	                #sFB_PECUpdate_380(iUDT_PECUpdateConfiguration := #iUDT_Configuration."380".PEC_Eos,
	                                   iUDT_ConveyorCommonConfiguration := #iUDT_Configuration."380".Conveyor.Common,
	                                   ix_PEC := #iUDT_MotorInput380.AllSensorPortInputs.LeftSensor,
	                                   ix_TeachingMode := FALSE,
	                                   qUDT_Status => #iqUDT_WorkstationStatus."380".PEC_Eos,
	                                   qi_GINwrite => #ti_dummy,
	                                   qx_PECFiltered => #tx_dummy,
	                                   iqa_TrackingData := #sa_TrackingArray_380,
	                                   iqUDT_ConveyorInterface := #sUDT_Interface_380,
	                                   iqUDT_UnknownGINRange := #iqUDT_UnknownGINRange,
	                                   iqUDT_FifoHeader := "DB_FIFOLostGIN".Header,
	                                   iqa_FifoData := "DB_FIFOLostGIN".Data,
	                                   iqUDT_Statistics := #iqUDT_WorkstationStatistics."380".PEC_Eos);

	            END_REGION

	            REGION Conveyor

	                #sUDT_Handshake_380.RTR := #iqUDT_WorkstationStatus."380".PEC_Eos.PEC;

	                #sFB_Conveyor_380(iUDT_ConveyorConfiguration := #iUDT_Configuration."380".Conveyor,
	                                  idi_PECEoSDistance := #iUDT_Configuration."380".PEC_Eos.Distance,
	                                  idi_PECBoSDistance := 0,
	                                  ii_ExternalSpeed := 0,
	                                  ix_SafetyOk := #ix_SafetyOk,
	                                  ix_24vOk := #ix_24vOk,
	                                  ix_400vOk := #ix_400vOk,
	                                  ix_HardwareOk := #ix_HardwareOk,
	                                  ix_ReverseDirection := #sx_DirectionChange380,
	                                  ix_PECEoS := #iqUDT_WorkstationStatus."380".PEC_Eos.PEC,
	                                  ix_PECBoS := TRUE,
	                                  ix_ExternalRequestHold := false,
	                                  qUDT_HMIStatus => #iqUDT_WorkstationStatus."380".Conveyor,
	                                  qUDT_Status => #iqUDT_WorkstationCommonStatus."380",
	                                  iqUDT_EquipmentControl := #iqUDT_EquipmentControl,
	                                  iqUDT_ConveyorCommand := #iqUDT_WorkstationCommands."380".Conveyor,
	                                  iqUDT_ConveyorInterface := #sUDT_Interface_380,
	                                  iqUDT_HandShakeUp := #sUDT_Handshake_360,
	                                  iqUDT_HandShake := #sUDT_Handshake_380,
	                                  iqUDT_Statistics := #iqUDT_WorkstationStatistics."380".Conveyor);
	            END_REGION

	            REGION MCO
	                #sFB_MCOConveyLinxAixController_380(iUDT_AixConfig := #iUDT_Configuration."380".MCO_M01,
	                                                    iv_AixInputsModule := #iUDT_MotorInput380,
	                                                    ix_24vOk := #ix_24vOk,
	                                                    ix_SimulationModeActive := "DB_Memory".Simulation,
	                                                    ii_MotorPositionId := 1,
	                                                    qUDT_HMIStatus => #iqUDT_WorkstationStatus."380".MCO_M01,
	                                                    iqv_AixOutputsModule := #qUDT_MotorOutput380,
	                                                    iqUDT_ConveyorInterface := #sUDT_Interface_380,
	                                                    iqUDT_MCOStatistics := #iqUDT_WorkstationStatistics."380".MCO_M01);
	            END_REGION


	        END_REGION

	        REGION 390

	            REGION Displacement

	                #sFB_Displacement390(#sUDT_Interface_390);

	            END_REGION

	            REGION Tracking

	                #sFB_Tracking_390(iUDT_ConveyorCommonConfiguration := #iUDT_Configuration."390".Conveyor.Common,
	                                  iqa_TrackingData := #sa_TrackingArray_390,
	                                  iqUDT_ConveyorInterface := #sUDT_Interface_390,
	                                  iqUDT_HandshakeUp := #sUDT_Handshake_370,
	                                  iqUDT_Handshake := #sUDT_Handshake_390);
	            END_REGION

	            REGION EOS

	                #sFB_PECUpdate_390(iUDT_PECUpdateConfiguration := #iUDT_Configuration."390".PEC_Eos,
	                                   iUDT_ConveyorCommonConfiguration := #iUDT_Configuration."390".Conveyor.Common,
	                                   ix_PEC := #iUDT_MotorInput390.AllSensorPortInputs.LeftSensor,
	                                   ix_TeachingMode := FALSE,
	                                   qUDT_Status => #iqUDT_WorkstationStatus."390".PEC_Eos,
	                                   qi_GINwrite => #ti_dummy,
	                                   qx_PECFiltered => #tx_dummy,
	                                   iqa_TrackingData := #sa_TrackingArray_390,
	                                   iqUDT_ConveyorInterface := #sUDT_Interface_390,
	                                   iqUDT_UnknownGINRange := #iqUDT_UnknownGINRange,
	                                   iqUDT_FifoHeader := "DB_FIFOLostGIN".Header,
	                                   iqa_FifoData := "DB_FIFOLostGIN".Data,
	                                   iqUDT_Statistics := #iqUDT_WorkstationStatistics."390".PEC_Eos);

	            END_REGION

	            REGION Conveyor

	                #sUDT_Handshake_390.RTR := #iqUDT_WorkstationStatus."390".PEC_Eos.PEC;


	                #sFB_Conveyor_390(iUDT_ConveyorConfiguration := #iUDT_Configuration."390".Conveyor,
	                                  idi_PECEoSDistance := #iUDT_Configuration."390".PEC_Eos.Distance,
	                                  idi_PECBoSDistance := 0,
	                                  ii_ExternalSpeed := 0,
	                                  ix_SafetyOk := #ix_SafetyOk,
	                                  ix_24vOk := #ix_24vOk,
	                                  ix_400vOk := #ix_400vOk,
	                                  ix_HardwareOk := #ix_HardwareOk,
	                                  ix_ReverseDirection := #sx_DirectionChange390,
	                                  ix_PECEoS := #iqUDT_WorkstationStatus."390".PEC_Eos.PEC,
	                                  ix_PECBoS := TRUE,
	                                  ix_ExternalRequestHold := FALSE,
	                                  qUDT_HMIStatus => #iqUDT_WorkstationStatus."390".Conveyor,
	                                  qUDT_Status => #iqUDT_WorkstationCommonStatus."390",
	                                  iqUDT_EquipmentControl := #iqUDT_EquipmentControl,
	                                  iqUDT_ConveyorCommand := #iqUDT_WorkstationCommands."390".Conveyor,
	                                  iqUDT_ConveyorInterface := #sUDT_Interface_390,
	                                  iqUDT_HandShakeUp := #sUDT_Handshake_370,
	                                  iqUDT_HandShake := #sUDT_Handshake_390,
	                                  iqUDT_Statistics := #iqUDT_WorkstationStatistics."390".Conveyor);
	            END_REGION

	            REGION MCO
	                #sFB_MCOConveyLinxAixController_390(iUDT_AixConfig := #iUDT_Configuration."390".MCO_M01,
	                                                    iv_AixInputsModule := #iUDT_MotorInput390,
	                                                    ix_24vOk := #ix_24vOk,
	                                                    ix_SimulationModeActive := "DB_Memory".Simulation,
	                                                    ii_MotorPositionId := 1,
	                                                    qUDT_HMIStatus => #iqUDT_WorkstationStatus."390".MCO_M01,
	                                                    iqv_AixOutputsModule := #qUDT_MotorOutput390,
	                                                    iqUDT_ConveyorInterface := #sUDT_Interface_390,
	                                                    iqUDT_MCOStatistics := #iqUDT_WorkstationStatistics."390".MCO_M01);
	            END_REGION


	        END_REGION
	        REGION 230

	            REGION Displacement

	                #sFB_Displacement230(#sUDT_Interface_230);

	            END_REGION

	            REGION Tracking

	                #sFB_Tracking_230(iUDT_ConveyorCommonConfiguration := #iUDT_Configuration."230".Conveyor.Common,
	                                  iqa_TrackingData := #sa_TrackingArray_230,
	                                  iqUDT_ConveyorInterface := #sUDT_Interface_230,
	                                  iqUDT_HandshakeUp := #sUDT_Handshake_230,
	                                  iqUDT_Handshake := #sUDT_Handshake_230);
	            END_REGION

	            REGION EOS

	                #sFB_PECUpdate_230(iUDT_PECUpdateConfiguration := #iUDT_Configuration."230".PEC_Eos,
	                                   iUDT_ConveyorCommonConfiguration := #iUDT_Configuration."230".Conveyor.Common,
	                                   ix_PEC := #iUDT_MotorInput230.AllSensorPortInputs.LeftSensor,
	                                   ix_TeachingMode := FALSE,
	                                   qUDT_Status => #iqUDT_WorkstationStatus."230".PEC_Eos,
	                                   qi_GINwrite => #ti_dummy,
	                                   qx_PECFiltered => #tx_dummy,
	                                   iqa_TrackingData := #sa_TrackingArray_230,
	                                   iqUDT_ConveyorInterface := #sUDT_Interface_230,
	                                   iqUDT_UnknownGINRange := #iqUDT_UnknownGINRange,
	                                   iqUDT_FifoHeader := "DB_FIFOLostGIN".Header,
	                                   iqa_FifoData := "DB_FIFOLostGIN".Data,
	                                   iqUDT_Statistics := #iqUDT_WorkstationStatistics."230".PEC_Eos);

	            END_REGION

	            REGION Conveyor
	                #sUDT_Handshake_230.RTR := #sUDT_Handshake_230.RTR OR #iqUDT_WorkstationStatus."230".PEC_Eos.PEC;

	                #sFB_Conveyor_230(iUDT_ConveyorConfiguration := #iUDT_Configuration."230".Conveyor,
	                                  idi_PECEoSDistance := #iUDT_Configuration."230".PEC_Eos.Distance,
	                                  idi_PECBoSDistance := 0,
	                                  ii_ExternalSpeed := 0,
	                                  ix_SafetyOk := #ix_SafetyOk,
	                                  ix_24vOk := #ix_24vOk,
	                                  ix_400vOk := #ix_400vOk,
	                                  ix_HardwareOk := #ix_HardwareOk,
	                                  ix_PECEoS := #iqUDT_WorkstationStatus."230".PEC_Eos.PEC,
	                                  ix_PECBoS := TRUE,
	                                  ix_ExternalRequestHold := #sx_Hold230,
	                                  qUDT_HMIStatus => #iqUDT_WorkstationStatus."230".Conveyor,
	                                  qUDT_Status => #iqUDT_WorkstationCommonStatus."230",
	                                  iqUDT_EquipmentControl := #iqUDT_EquipmentControl,
	                                  iqUDT_ConveyorCommand := #iqUDT_WorkstationCommands."230".Conveyor,
	                                  iqUDT_ConveyorInterface := #sUDT_Interface_230,
	                                  iqUDT_HandShakeUp := #sUDT_Handshake_230,
	                                  iqUDT_HandShake := #sUDT_Handshake_230,
	                                  iqUDT_Statistics := #iqUDT_WorkstationStatistics."230".Conveyor);
	            END_REGION

	            REGION MCO
	                #sFB_MCOConveyLinxAixController_230(iUDT_AixConfig := #iUDT_Configuration."230".MCO_M01,
	                                                    iv_AixInputsModule := #iUDT_MotorInput230,
	                                                    ix_24vOk := #ix_24vOk,
	                                                    ix_SimulationModeActive := "DB_Memory".Simulation,
	                                                    ii_MotorPositionId := 1,
	                                                    qUDT_HMIStatus => #iqUDT_WorkstationStatus."230".MCO_M01,
	                                                    iqv_AixOutputsModule := #qUDT_MotorOutput230,
	                                                    iqUDT_ConveyorInterface := #sUDT_Interface_230,
	                                                    iqUDT_MCOStatistics := #iqUDT_WorkstationStatistics."230".MCO_M01);
	            END_REGION

	        END_REGION

	        REGION 240

	            REGION Displacement

	                #sFB_Displacement240(#sUDT_Interface_240);

	            END_REGION

	            REGION MCO
	                #sFB_MCOConveyLinxAixController_240(iUDT_AixConfig := #iUDT_Configuration."240".MCO_M01,
	                                                    iv_AixInputsModule := #iUDT_MotorInput240,
	                                                    ii_PositionSetpoint := #iqUDT_RATPositioning240.Lower.EndPosition,
	                                                    ix_24vOk := #ix_24vOk,
	                                                    ix_SimulationModeActive := "DB_Memory".Simulation,
	                                                    ii_MotorPositionId := 1,
	                                                    ix_StartPositioning := #iqUDT_RATPositioning240.Lower.Start,
	                                                    ix_ResetPosition := #iqUDT_RATPositioning240.Lower.ResetPosition,
	                                                    qUDT_HMIStatus => #iqUDT_WorkstationStatus."240".MCO_M01,
	                                                    qx_Positioned => #iqUDT_RATPositioning240.Lower.Done,
	                                                    iqv_AixOutputsModule := #qUDT_MotorOutput240,
	                                                    iqUDT_ConveyorInterface := #sUDT_Interface_240,
	                                                    iqUDT_MCOStatistics := #iqUDT_WorkstationStatistics."240".MCO_M01);
	            END_REGION


	        END_REGION

	        REGION 241

	            REGION Displacement

	                #sFB_Displacement241(#sUDT_Interface_241);

	            END_REGION

	            REGION RAT

	                #sFB_RightAngledTransfer_241(iUDT_Configuration := #iUDT_Configuration."241".RightAngledTransfer,
	                                             iUDT_LowerConveyorConfiguration := #iUDT_Configuration."240".Conveyor,
	                                             iUDT_UpperConveyorConfiguration := #iUDT_Configuration."241".Conveyor,
	                                             iUDT_PECConfiguration := #iUDT_Configuration."240".PEC_Eos,
	                                             ii_DestinationA := #si_240DestinationA,
	                                             ii_DestinationB := #si_240DestinationB,
	                                             ii_DestinationC := #si_240DestinationC,
	                                             ii_DestinationD := #si_240DestinationD,
	                                             ix_HardwareOk := #ix_HardwareOk,
	                                             ix_400vOk := #ix_400vOk,
	                                             ix_24vOk := #ix_24vOk,
	                                             ix_SafetyOk := #ix_SafetyOk,
	                                             ix_AirPressureOk := #ix_AirPressureOk,
	                                             ix_SectionIsDown := #ix_SectionIsDown241,
	                                             ix_SectionIsUp := #ix_SectionIsUp241,
	                                             ix_ConveyorAAuto := #iqUDT_WorkstationCommonStatus."230".AutoON,
	                                             ix_ConveyorBAuto := #iqUDT_WorkstationCommonStatus."250".AutoON,
	                                             ix_ConveyorCAuto := FALSE,
	                                             ix_ConveyorDAuto := #iqUDT_WorkstationCommonStatus."370".AutoON,
	                                             ix_PEC := #iUDT_MotorInput240.AllSensorPortInputs.LeftSensor,
	                                             ix_ExternalReceiveRequestA := NOT #iqUDT_WorkstationStatus."230".PEC_Eos.PEC AND NOT #sx_TransferOut380 AND NOT #sx_TransferOut390,
	                                             ix_ExternalReceiveRequestB := false,
	                                             ix_ExternalReceiveRequestC := false,
	                                             ix_ExternalReceiveRequestD := #sFB_RightAngledTransfer_371.qx_ExternalSendRequestD,//NOT #iUDT_MotorInput370.AllSensorPortInputs.LeftSensor AND (#sx_TransferOut380 OR #sx_TransferOut390 OR #iqx_ClearRightStation),,
	                                             ix_PECInfeedA := #iqUDT_WorkstationStatus."230".PEC_Eos.PEC,
	                                             ix_PECInfeedD := #iqUDT_WorkstationStatus."370".PEC_Eos.PEC,
	                                             qUDT_HMIRATStatus => #iqUDT_WorkstationStatus."241".RightAngledTransfer,
	                                             qUDT_HMIConveyorStatus => #iqUDT_WorkstationStatus."240".Conveyor,
	                                             qUDT_HMIPECStatus => #iqUDT_WorkstationStatus."240".PEC_Eos,
	                                             qUDT_RATStatus => #iqUDT_WorkstationCommonStatus."241",
	                                             qUDT_ConveyorStatus => #iqUDT_WorkstationCommonStatus."240",
	                                             qx_PopupControl => #qx_PopupControl241,
	                                             iqUDT_EquipmentControl := #iqUDT_EquipmentControl,
	                                             iqUDT_RATCommand := #iqUDT_WorkstationCommands."241".RightAngledTransfer,
	                                             iqUDT_ConveyorCommand := #iqUDT_WorkstationCommands."240".Conveyor,
	                                             iqUDT_RATStatistics := #iqUDT_WorkstationStatistics."241".RightAngledTransfer,
	                                             iqUDT_ConveyorStatistics := #iqUDT_WorkstationStatistics."240".Conveyor,
	                                             iqUDT_PECStatistics := #iqUDT_WorkstationStatistics."240".PEC_Eos,
	                                             iqUDT_HandShakeConveyorA := #sUDT_Handshake_230,
	                                             iqUDT_HandShakeConveyorB := #sUDT_Handshake_240,
	                                             iqUDT_HandShakeConveyorC := #sUDT_Handshake_241,
	                                             iqUDT_HandShakeConveyorD := #sUDT_Handshake_371,
	                                             iqUDT_LowerConveyorInterface := #sUDT_Interface_240,
	                                             iqUDT_UpperConveyorInterface := #sUDT_Interface_241,
	                                             iqUDT_RATPositioning := #iqUDT_RATPositioning240,
	                                             iqUDT_BladeStopEoSInterface := #tUDT_DummyBladeStop,
	                                             iqUDT_BladeStopBoSInterface := #tUDT_DummyBladeStop);

	            END_REGION

	            REGION MCO
	                #sFB_MCOConveyLinxAixController_241(iUDT_AixConfig := #iUDT_Configuration."241".MCO_M01,
	                                                    iv_AixInputsModule := #iUDT_MotorInput240,
	                                                    ii_PositionSetpoint := #iqUDT_RATPositioning240.Upper.EndPosition,
	                                                    ix_24vOk := #ix_24vOk,
	                                                    ix_SimulationModeActive := "DB_Memory".Simulation,
	                                                    ii_MotorPositionId := 2,
	                                                    ix_StartPositioning := #iqUDT_RATPositioning240.Upper.Start,
	                                                    ix_ResetPosition := #iqUDT_RATPositioning240.Upper.ResetPosition,
	                                                    qUDT_HMIStatus => #iqUDT_WorkstationStatus."241".MCO_M01,
	                                                    qx_Positioned => #iqUDT_RATPositioning240.Upper.Done,
	                                                    iqv_AixOutputsModule := #qUDT_MotorOutput240,
	                                                    iqUDT_ConveyorInterface := #sUDT_Interface_241,
	                                                    iqUDT_MCOStatistics := #iqUDT_WorkstationStatistics."241".MCO_M01);
	            END_REGION
	        END_REGION

	        REGION 250

	            REGION Displacement

	                #sFB_Displacement250(#sUDT_Interface_250);

	            END_REGION

	            REGION EOS

	                #sFB_PECUpdate_250(iUDT_PECUpdateConfiguration := #iUDT_Configuration."250".PEC_EoS,
	                                   iUDT_ConveyorCommonConfiguration := #iUDT_Configuration."250".Conveyor.Common,
	                                   ix_PEC := #iUDT_MotorInput250.AllSensorPortInputs.LeftSensor,
	                                   ix_TeachingMode := FALSE,
	                                   qUDT_Status => #iqUDT_WorkstationStatus."250".PEC_EoS,
	                                   qi_GINwrite => #ti_dummy,
	                                   qx_PECFiltered => #tx_dummy,
	                                   iqa_TrackingData := #sa_TrackingArray_250,
	                                   iqUDT_ConveyorInterface := #sUDT_Interface_250,
	                                   iqUDT_UnknownGINRange := #iqUDT_UnknownGINRange,
	                                   iqUDT_FifoHeader := "DB_FIFOLostGIN".Header,
	                                   iqa_FifoData := "DB_FIFOLostGIN".Data,
	                                   iqUDT_Statistics := #iqUDT_WorkstationStatistics."250".PEC_EoS);

	            END_REGION

	            REGION Conveyor

	                #sUDT_Handshake_250.RTR := #sUDT_Handshake_250.RTR OR #iqUDT_WorkstationStatus."250".PEC_EoS.PEC;

	                #sFB_Conveyor_250(iUDT_ConveyorConfiguration := #iUDT_Configuration."250".Conveyor,
	                                  idi_PECEoSDistance := #iUDT_Configuration."250".PEC_EoS.Distance,
	                                  idi_PECBoSDistance := 0,
	                                  ii_ExternalSpeed := 0,
	                                  ix_SafetyOk := #ix_SafetyOk,
	                                  ix_24vOk := #ix_24vOk,
	                                  ix_400vOk := #ix_400vOk,
	                                  ix_HardwareOk := #ix_HardwareOk,
	                                  ix_PECEoS := #iqUDT_WorkstationStatus."250".PEC_EoS.PEC,
	                                  ix_PECBoS := TRUE,
	                                  ix_ExternalRequestHold := false,
	                                  qUDT_HMIStatus => #iqUDT_WorkstationStatus."250".Conveyor,
	                                  qUDT_Status => #iqUDT_WorkstationCommonStatus."250",
	                                  iqUDT_EquipmentControl := #iqUDT_EquipmentControl,
	                                  iqUDT_ConveyorCommand := #iqUDT_WorkstationCommands."250".Conveyor,
	                                  iqUDT_ConveyorInterface := #sUDT_Interface_250,
	                                  iqUDT_HandShakeUp := #sUDT_Handshake_240,
	                                  iqUDT_HandShake := #sUDT_Handshake_250,
	                                  iqUDT_Statistics := #iqUDT_WorkstationStatistics."250".Conveyor);
	            END_REGION

	            REGION MCO
	                #sFB_MCOConveyLinxAixController_250(iUDT_AixConfig := #iUDT_Configuration."250".MCO_M01,
	                                                    iv_AixInputsModule := #iUDT_MotorInput250,
	                                                    ix_24vOk := #ix_24vOk,
	                                                    ix_SimulationModeActive := "DB_Memory".Simulation,
	                                                    ii_MotorPositionId := 1,
	                                                    qUDT_HMIStatus => #iqUDT_WorkstationStatus."250".MCO_M01,
	                                                    iqv_AixOutputsModule := #qUDT_MotorOutput250,
	                                                    iqUDT_ConveyorInterface := #sUDT_Interface_250,
	                                                    iqUDT_MCOStatistics := #iqUDT_WorkstationStatistics."250".MCO_M01);
	            END_REGION


	        END_REGION

	        REGION 260


	            REGION Displacement

	                #sFB_Displacement260(#sUDT_Interface_260);

	            END_REGION

	            REGION Conveyor
	                #sFB_Conveyor_260(iUDT_ConveyorConfiguration := #iUDT_Configuration."260".Conveyor,
	                                  idi_PECEoSDistance := 0,
	                                  idi_PECBoSDistance := 0,
	                                  ii_ExternalSpeed := 0,
	                                  ix_SafetyOk := #ix_SafetyOk,
	                                  ix_24vOk := #ix_24vOk,
	                                  ix_400vOk := #ix_400vOk,
	                                  ix_HardwareOk := #ix_HardwareOk,
	                                  ix_PECEoS := TRUE,
	                                  ix_PECBoS := TRUE,
	                                  ix_ExternalRequestHold := false,
	                                  qUDT_HMIStatus => #iqUDT_WorkstationStatus."260".Conveyor,
	                                  qUDT_Status => #iqUDT_WorkstationCommonStatus."260",
	                                  iqUDT_EquipmentControl := #iqUDT_EquipmentControl,
	                                  iqUDT_ConveyorCommand := #iqUDT_WorkstationCommands."260".Conveyor,
	                                  iqUDT_ConveyorInterface := #sUDT_Interface_260,
	                                  iqUDT_HandShakeUp := #sUDT_Handshake_250,
	                                  iqUDT_HandShake := #sUDT_Handshake_260,
	                                  iqUDT_Statistics := #iqUDT_WorkstationStatistics."260".Conveyor);
	            END_REGION

	            REGION VFD

	                #sFB_VfdNORDPPO4_260(iUDT_VFDConfig := #iUDT_Configuration."260".VFD,
	                                     iUDT_VFDInputs := #iUDT_MotorInput260,
	                                     iUDT_MotorData := #iUDT_MotorData260,
	                                     ix_24vOk := #ix_24vOk,
	                                     ix_400vOk := #ix_400vOk,
	                                     ix_QuickStopDisable := TRUE,
	                                     ix_SimulationModeActive := "DB_Memory".Simulation,
	                                     qUDT_HMIStatus => #iqUDT_WorkstationStatus."260".VFD,
	                                     qUDT_VFDOutputs => #qUDT_MotorOutput260,
	                                     iqUDT_ConveyorInterface := #sUDT_Interface_260,
	                                     iqUDT_VFDStatistics := #iqUDT_WorkstationStatistics."260".VFD,
	                                     iqx_StartCommissioning := #iqx_StartComissioning260);

	            END_REGION


	        END_REGION

	        REGION 270

	            REGION Displacement

	                #sFB_Displacement270(#sUDT_Interface_270);

	            END_REGION

	            REGION EoS

	                #sFB_PEC_270(ix_PEC := #iUDT_MotorInput270.AllSensorPortInputs.LeftSensor,
	                             iUDT_PECConfiguration := #iUDT_Configuration."270".PEC_EoS,
	                             qUDT_HMIStatus => #iqUDT_WorkstationStatus."270".PEC_EoS,
	                             iqUDT_ConveyorInterface := #sUDT_Interface_270,
	                             iqUDT_PECStatistics := #iqUDT_WorkstationStatistics."270".PEC_EoS);

	            END_REGION

	            REGION Conveyor
	                #sFB_Conveyor_270(iUDT_ConveyorConfiguration := #iUDT_Configuration."270".Conveyor,
	                                  idi_PECEoSDistance := #iUDT_Configuration."270".PEC_EoS.Distance,
	                                  idi_PECBoSDistance := 0,
	                                  ii_ExternalSpeed := 0,
	                                  ix_SafetyOk := #ix_SafetyOk,
	                                  ix_24vOk := #ix_24vOk,
	                                  ix_400vOk := #ix_400vOk,
	                                  ix_HardwareOk := #ix_HardwareOk,
	                                  ix_PECEoS := #iqUDT_WorkstationStatus."270".PEC_EoS.PEC,
	                                  ix_PECBoS := TRUE,
	                                  ix_ExternalRequestHold := false,
	                                  qUDT_HMIStatus => #iqUDT_WorkstationStatus."270".Conveyor,
	                                  qUDT_Status => #iqUDT_WorkstationCommonStatus."270",
	                                  iqUDT_EquipmentControl := #iqUDT_EquipmentControl,
	                                  iqUDT_ConveyorCommand := #iqUDT_WorkstationCommands."270".Conveyor,
	                                  iqUDT_ConveyorInterface := #sUDT_Interface_270,
	                                  iqUDT_HandShakeUp := #sUDT_Handshake_260,
	                                  iqUDT_HandShake := #sUDT_Handshake_270,
	                                  iqUDT_Statistics := #iqUDT_WorkstationStatistics."270".Conveyor);
	            END_REGION

	            REGION MCO
	                #sFB_MCOConveyLinxAixController_270(iUDT_AixConfig := #iUDT_Configuration."270".MCO_M01,
	                                                    iv_AixInputsModule := #iUDT_MotorInput270,
	                                                    ix_24vOk := #ix_24vOk,
	                                                    ix_SimulationModeActive := "DB_Memory".Simulation,
	                                                    ii_MotorPositionId := 1,
	                                                    qUDT_HMIStatus => #iqUDT_WorkstationStatus."270".MCO_M01,
	                                                    iqv_AixOutputsModule := #qUDT_MotorOutput270,
	                                                    iqUDT_ConveyorInterface := #sUDT_Interface_270,
	                                                    iqUDT_MCOStatistics := #iqUDT_WorkstationStatistics."270".MCO_M01);
	            END_REGION
	        END_REGION

	        REGION 280

	            REGION Displacement

	                #sFB_Displacement280(#sUDT_Interface_280);

	            END_REGION

	            REGION EoS

	                #sFB_PEC_280(ix_PEC := #iUDT_MotorInput270.AllSensorPortInputs.RightSensor,
	                             iUDT_PECConfiguration := #iUDT_Configuration."280".PEC_EoS,
	                             qUDT_HMIStatus => #iqUDT_WorkstationStatus."280".PEC_EoS,
	                             iqUDT_ConveyorInterface := #sUDT_Interface_280,
	                             iqUDT_PECStatistics := #iqUDT_WorkstationStatistics."280".PEC_EoS);

	            END_REGION

	            REGION Conveyor
	                #iqUDT_HandshakeDownstream280.RTR := #iqUDT_HandshakeDownstream280.RTR OR #iqUDT_WorkstationStatus."280".PEC_EoS.PEC;
	                #sFB_Conveyor_280(iUDT_ConveyorConfiguration := #iUDT_Configuration."280".Conveyor,
	                                  idi_PECEoSDistance := #iUDT_Configuration."280".PEC_EoS.Distance,
	                                  idi_PECBoSDistance := 0,
	                                  ii_ExternalSpeed := 0,
	                                  ix_SafetyOk := #ix_SafetyOk,
	                                  ix_24vOk := #ix_24vOk,
	                                  ix_400vOk := #ix_400vOk,
	                                  ix_HardwareOk := #ix_HardwareOk,
	                                  ix_PECEoS := #iqUDT_WorkstationStatus."280".PEC_EoS.PEC,
	                                  ix_PECBoS := TRUE,
	                                  ix_ExternalRequestHold := false,
	                                  qUDT_HMIStatus => #iqUDT_WorkstationStatus."280".Conveyor,
	                                  qUDT_Status => #iqUDT_WorkstationCommonStatus."280",
	                                  iqUDT_EquipmentControl := #iqUDT_EquipmentControl,
	                                  iqUDT_ConveyorCommand := #iqUDT_WorkstationCommands."280".Conveyor,
	                                  iqUDT_ConveyorInterface := #sUDT_Interface_280,
	                                  iqUDT_HandShakeUp := #sUDT_Handshake_270,
	                                  iqUDT_HandShake := #iqUDT_HandshakeDownstream280,
	                                  iqUDT_Statistics := #iqUDT_WorkstationStatistics."280".Conveyor);
	            END_REGION
	            REGION MCO
	                #sFB_MCOConveyLinxAixController_280(iUDT_AixConfig := #iUDT_Configuration."280".MCO_M01,
	                                                    iv_AixInputsModule := #iUDT_MotorInput270,
	                                                    ix_24vOk := #ix_24vOk,
	                                                    ix_SimulationModeActive := "DB_Memory".Simulation,
	                                                    ii_MotorPositionId := 2,
	                                                    qUDT_HMIStatus => #iqUDT_WorkstationStatus."280".MCO_M01,
	                                                    iqv_AixOutputsModule := #qUDT_MotorOutput270,
	                                                    iqUDT_ConveyorInterface := #sUDT_Interface_280,
	                                                    iqUDT_MCOStatistics := #iqUDT_WorkstationStatistics."010".MCO_M01);
	            END_REGION
	        END_REGION
	    END_REGION
	END_IF;

	IF #iUDT_Configuration.GlobalConfig.LeftStationExists THEN
	    REGION Left Station
	        REGION Left Station Control

	            //Triggers
	            #s_F_Trig_540(CLK := #iqUDT_WorkstationStatus."540".PEC_Eos.PEC);
	            #s_F_Trig_ClearLeft(CLK := #sx_ClearLeftStation);

	            //If any request comes, start if possible
	            IF #iqUDT_WorkstationStatus."680".PEC_Eos.PEC
	                AND #ix_StationActive
	                AND NOT #sx_ActiveRequest680
	                AND NOT #sx_TransferOut680
	                AND NOT #sx_ClearLeftStation
	            THEN
	                #sx_ActiveRequest680 := TRUE;

	            END_IF;
	            IF #iqUDT_WorkstationStatus."690".PEC_Eos.PEC
	                AND #ix_StationActive
	                AND NOT #sx_ActiveRequest690
	                AND NOT #sx_TransferOut690
	                AND NOT #sx_ClearLeftStation
	            THEN
	                #sx_ActiveRequest690 := TRUE;
	            END_IF;

	            //Request in progress
	            IF #sx_ActiveRequest680 AND #sFB_RightAngledTransfer_651.qx_ExternalSendRequestB THEN
	                #sx_ReqInProgress680 := TRUE;
	            END_IF;

	            IF #sx_ActiveRequest690 AND #sFB_RightAngledTransfer_641.qx_ExternalSendRequestB THEN
	                #sx_ReqInProgress690 := TRUE;
	            END_IF;

	            //Request fulfilled
	            IF #sx_ActiveRequest690 AND NOT #iqUDT_WorkstationStatus."690".PEC_Eos.PEC
	            THEN
	                #sx_ActiveRequest690 := FALSE;
	                #sx_ReqInProgress690 := FALSE;
	            END_IF;

	            IF #sx_ActiveRequest680 AND NOT #iqUDT_WorkstationStatus."680".PEC_Eos.PEC
	            THEN
	                #sx_ActiveRequest680 := FALSE;
	                #sx_ReqInProgress680 := FALSE;
	            END_IF;

	            //Start transfering out
	            IF #iqx_Done680
	                AND NOT #sx_TransferOut690
	                AND (#iqUDT_WorkstationStatus."540".PEC_Eos.PEC OR #sx_Hold530)
	                AND NOT #iqUDT_WorkstationStatus."680".PEC_Eos.PEC
	            THEN
	                #sx_TransferOut680 := TRUE;
	                #sx_Hold530 := TRUE;
	                #iqx_Done680 := FALSE;
	            END_IF;

	            IF #iqx_Done690
	                AND NOT #sx_TransferOut680
	                AND (#iqUDT_WorkstationStatus."540".PEC_Eos.PEC OR #sx_Hold530)
	                AND NOT #iqUDT_WorkstationStatus."690".PEC_Eos.PEC
	            THEN
	                #sx_TransferOut690 := TRUE;
	                #sx_Hold530 := TRUE;
	                #iqx_Done690 := FALSE;
	            END_IF;

	            //If transfer is in progress, set up directions and destinations

	            IF #sx_TransferOut680 THEN
	                #sx_DirectionChange680 := TRUE;
	            END_IF;

	            IF #sx_TransferOut690 THEN
	                #sx_DirectionChange690 := TRUE;
	            END_IF;

	            //If transfer is over set up directions and destinations
	            IF NOT #sx_TransferOut680 AND NOT #sx_TransferOut690 THEN
	                #sx_Hold530 := FALSE;
	            END_IF;

	            IF #sx_TransferOut680 AND #s_F_Trig_540.Q
	            THEN
	                #sx_TransferOut680 := FALSE;
	                #sx_DirectionChange680 := FALSE;
	            END_IF;

	            IF #sx_TransferOut690 AND #s_F_Trig_540.Q
	            THEN
	                #sx_TransferOut690 := FALSE;
	                #sx_DirectionChange690 := FALSE;
	            END_IF;

	            //Destinations from RAT 640
	            IF #sx_ActiveRequest690 AND NOT #sx_ReqInProgress690 THEN
	                #si_640DestinationA := 1;
	                #si_640DestinationB := 0;
	                #si_640DestinationC := 0;
	                #si_640DestinationD := 0;

	            ELSIF #iqUDT_WorkstationStatus."650".PEC_Eos.PEC THEN
	                #si_640DestinationA := 2;
	                #si_640DestinationB := 0;
	                #si_640DestinationC := 0;
	                #si_640DestinationD := 0;
	            ELSE
	                #si_640DestinationA := 0;
	                #si_640DestinationB := 0;
	                #si_640DestinationC := 0;
	                #si_640DestinationD := 0;
	            END_IF;


	            //Destinations from RAT 650
	            IF #sx_ActiveRequest680 AND NOT #sx_ReqInProgress380 THEN
	                #si_650DestinationA := 0;
	                #si_650DestinationB := 0;
	                #si_650DestinationC := 1;
	                #si_650DestinationD := 0;
	            ELSE

	                #si_650DestinationA := 0;
	                #si_650DestinationB := 0;
	                #si_650DestinationC := 0;
	                #si_650DestinationD := 0;
	            END_IF;

	            //Other destinations (stay the same as long as station is operating)
	            #si_540DestinationA := 1;
	            #si_540DestinationB := 0;
	            #si_540DestinationC := 1;
	            #si_540DestinationD := 0;

	            #si_660DestinationA := 1;
	            #si_660DestinationB := 2;
	            #si_660DestinationC := 0;
	            #si_660DestinationD := 0;

	            #si_670DestinationA := 1;
	            #si_670DestinationB := 2;
	            #si_670DestinationC := 0;
	            #si_670DestinationD := 2;

	        END_REGION
	        REGION Clear Left Station
	            //When clearing procedure is requested, set directions and destinations
	            IF NOT #ix_LeftStationActive THEN

	                #sx_ClearLeftStation := TRUE;

	                #sx_DirectionChange680 := TRUE;
	                #sx_DirectionChange690 := TRUE;

	                #si_640DestinationA := 1;
	                #si_640DestinationB := 0;
	                #si_640DestinationC := 0;
	                #si_640DestinationD := 0;

	                #si_650DestinationA := 0;
	                #si_650DestinationB := 0;
	                #si_650DestinationC := 1;
	                #si_650DestinationD := 0;

	                #si_660DestinationA := 2;
	                #si_660DestinationB := 2;
	                #si_660DestinationC := 0;
	                #si_660DestinationD := 0;

	                #si_670DestinationA := 2;
	                #si_670DestinationB := 2;
	                #si_670DestinationC := 0;
	                #si_670DestinationD := 2;
	            ELSE
	                #sx_ClearLeftStation := FALSE;
	            END_IF;
	            //When clearing procedure is done reset directions
	            IF #s_F_Trig_ClearLeft.Q THEN
	                #sx_DirectionChange680 := FALSE;
	                #sx_DirectionChange690 := FALSE;
	            END_IF;

	        END_REGION

	        REGION 610


	            REGION Displacement

	                #sFB_Displacement610(#sUDT_Interface_610);

	            END_REGION


	            REGION Conveyor
	                #sFB_Conveyor_610(iUDT_ConveyorConfiguration := #iUDT_Configuration."610".Conveyor,
	                                  idi_PECEoSDistance := 0,
	                                  idi_PECBoSDistance := 0,
	                                  ii_ExternalSpeed := 0,
	                                  ix_SafetyOk := #ix_SafetyOk,
	                                  ix_24vOk := #ix_24vOk,
	                                  ix_400vOk := #ix_400vOk,
	                                  ix_HardwareOk := #ix_HardwareOk,
	                                  ix_PECEoS := TRUE,
	                                  ix_PECBoS := TRUE,
	                                  ix_ExternalRequestHold := false,
	                                  qUDT_HMIStatus => #iqUDT_WorkstationStatus."610".Conveyor,
	                                  qUDT_Status => #iqUDT_WorkstationCommonStatus."610",
	                                  iqUDT_EquipmentControl := #iqUDT_EquipmentControl,
	                                  iqUDT_ConveyorCommand := #iqUDT_WorkstationCommands."610".Conveyor,
	                                  iqUDT_ConveyorInterface := #sUDT_Interface_610,
	                                  iqUDT_HandShakeUp := #iqUDT_HandshakeUpstream610,
	                                  iqUDT_HandShake := #sUDT_Handshake_610,
	                                  iqUDT_Statistics := #iqUDT_WorkstationStatistics."610".Conveyor);
	            END_REGION

	            REGION VFD

	                #sFB_VfdNORDPPO4_610(iUDT_VFDConfig := #iUDT_Configuration."610".VFD,
	                                     iUDT_VFDInputs := #iUDT_MotorInput610,
	                                     iUDT_MotorData := #iUDT_MotorData610,
	                                     ix_24vOk := #ix_24vOk,
	                                     ix_400vOk := #ix_400vOk,
	                                     ix_QuickStopDisable := TRUE,
	                                     ix_SimulationModeActive := "DB_Memory".Simulation,
	                                     qUDT_HMIStatus => #iqUDT_WorkstationStatus."610".VFD,
	                                     qUDT_VFDOutputs => #qUDT_MotorOutput610,
	                                     iqUDT_ConveyorInterface := #sUDT_Interface_610,
	                                     iqUDT_VFDStatistics := #iqUDT_WorkstationStatistics."610".VFD,
	                                     iqx_StartCommissioning := #iqx_StartComissioning610);


	            END_REGION
	        END_REGION


	        REGION 620

	            REGION Displacement

	                #sFB_Displacement620(#sUDT_Interface_620);

	            END_REGION

	            REGION Tracking

	                #sFB_Tracking_620(iUDT_ConveyorCommonConfiguration := #iUDT_Configuration."620".Conveyor.Common,
	                                  iqa_TrackingData := #sa_TrackingArray_620,
	                                  iqUDT_ConveyorInterface := #sUDT_Interface_620,
	                                  iqUDT_HandshakeUp := #sUDT_Handshake_610,
	                                  iqUDT_Handshake := #sUDT_Handshake_620);
	            END_REGION

	            REGION EOS

	                #sFB_PECUpdate_620(iUDT_PECUpdateConfiguration := #iUDT_Configuration."620".PEC_Eos,
	                                   iUDT_ConveyorCommonConfiguration := #iUDT_Configuration."620".Conveyor.Common,
	                                   ix_PEC := #iUDT_MotorInput620.AllSensorPortInputs.LeftSensor,
	                                   ix_TeachingMode := FALSE,
	                                   qUDT_Status => #iqUDT_WorkstationStatus."620".PEC_Eos,
	                                   qi_GINwrite => #ti_dummy,
	                                   qx_PECFiltered => #tx_dummy,
	                                   iqa_TrackingData := #sa_TrackingArray_620,
	                                   iqUDT_ConveyorInterface := #sUDT_Interface_620,
	                                   iqUDT_UnknownGINRange := #iqUDT_UnknownGINRange,
	                                   iqUDT_FifoHeader := "DB_FIFOLostGIN".Header,
	                                   iqa_FifoData := "DB_FIFOLostGIN".Data,
	                                   iqUDT_Statistics := #iqUDT_WorkstationStatistics."620".PEC_Eos);

	            END_REGION

	            REGION Conveyor
	                #sFB_Conveyor_620(iUDT_ConveyorConfiguration := #iUDT_Configuration."620".Conveyor,
	                                  idi_PECEoSDistance := #iUDT_Configuration."620".PEC_Eos.Distance,
	                                  idi_PECBoSDistance := 0,
	                                  ii_ExternalSpeed := 0,
	                                  ix_SafetyOk := #ix_SafetyOk,
	                                  ix_24vOk := #ix_24vOk,
	                                  ix_400vOk := #ix_400vOk,
	                                  ix_HardwareOk := #ix_HardwareOk,
	                                  ix_PECEoS := #iqUDT_WorkstationStatus."620".PEC_Eos.PEC,
	                                  ix_PECBoS := TRUE,
	                                  ix_ExternalRequestHold := FALSE,
	                                  qUDT_HMIStatus => #iqUDT_WorkstationStatus."620".Conveyor,
	                                  qUDT_Status => #iqUDT_WorkstationCommonStatus."620",
	                                  iqUDT_EquipmentControl := #iqUDT_EquipmentControl,
	                                  iqUDT_ConveyorCommand := #iqUDT_WorkstationCommands."620".Conveyor,
	                                  iqUDT_ConveyorInterface := #sUDT_Interface_620,
	                                  iqUDT_HandShakeUp := #sUDT_Handshake_610,
	                                  iqUDT_HandShake := #sUDT_Handshake_620,
	                                  iqUDT_Statistics := #iqUDT_WorkstationStatistics."620".Conveyor);
	            END_REGION

	            REGION MCO
	                #sFB_MCOConveyLinxAixController_620(iUDT_AixConfig := #iUDT_Configuration."620".MCO_M01,
	                                                    iv_AixInputsModule := #iUDT_MotorInput620,
	                                                    ix_24vOk := #ix_24vOk,
	                                                    ix_SimulationModeActive := "DB_Memory".Simulation,
	                                                    ii_MotorPositionId := 1,
	                                                    qUDT_HMIStatus => #iqUDT_WorkstationStatus."620".MCO_M01,
	                                                    iqv_AixOutputsModule := #qUDT_MotorOutput620,
	                                                    iqUDT_ConveyorInterface := #sUDT_Interface_620,
	                                                    iqUDT_MCOStatistics := #iqUDT_WorkstationStatistics."620".MCO_M01);
	            END_REGION


	        END_REGION

	        REGION 630

	            REGION Displacement

	                #sFB_Displacement630(#sUDT_Interface_630);

	            END_REGION

	            REGION Tracking

	                #sFB_Tracking_630(iUDT_ConveyorCommonConfiguration := #iUDT_Configuration."630".Conveyor.Common,
	                                  iqa_TrackingData := #sa_TrackingArray_630,
	                                  iqUDT_ConveyorInterface := #sUDT_Interface_630,
	                                  iqUDT_HandshakeUp := #sUDT_Handshake_620,
	                                  iqUDT_Handshake := #sUDT_Handshake_630);
	            END_REGION

	            REGION EOS

	                #sFB_PECUpdate_630(iUDT_PECUpdateConfiguration := #iUDT_Configuration."630".PEC_Eos,
	                                   iUDT_ConveyorCommonConfiguration := #iUDT_Configuration."630".Conveyor.Common,
	                                   ix_PEC := #iUDT_MotorInput620.AllSensorPortInputs.RightSensor,
	                                   ix_TeachingMode := FALSE,
	                                   qUDT_Status => #iqUDT_WorkstationStatus."630".PEC_Eos,
	                                   qi_GINwrite => #ti_dummy,
	                                   qx_PECFiltered => #tx_dummy,
	                                   iqa_TrackingData := #sa_TrackingArray_630,
	                                   iqUDT_ConveyorInterface := #sUDT_Interface_630,
	                                   iqUDT_UnknownGINRange := #iqUDT_UnknownGINRange,
	                                   iqUDT_FifoHeader := "DB_FIFOLostGIN".Header,
	                                   iqa_FifoData := "DB_FIFOLostGIN".Data,
	                                   iqUDT_Statistics := #iqUDT_WorkstationStatistics."630".PEC_Eos);

	            END_REGION

	            REGION Scanner

	                #sFB_CognexDM260_630(iUDT_CognexDM260_IN := #iUDT_ScannerInput630,
	                                     qs_Barcode => #ts_Barcode630,
	                                     iqUDT_EquipmentControl := #iqUDT_EquipmentControl,
	                                     ix_Trigger := #sa_TrackingArray_630[60] > 0,
	                                     qUDT_CognexDM260_OUT => #qUDT_ScannerOutput630,
	                                     qw_RetVal => #tw_dummy);

	            END_REGION

	            REGION Conveyor
	                #sUDT_Handshake_630.RTR := #sUDT_Handshake_630.RTR OR #iqUDT_WorkstationStatus."630".PEC_Eos.PEC;

	                #sFB_Conveyor_630(iUDT_ConveyorConfiguration := #iUDT_Configuration."630".Conveyor,
	                                  idi_PECEoSDistance := #iUDT_Configuration."630".PEC_Eos.Distance,
	                                  idi_PECBoSDistance := 0,
	                                  ii_ExternalSpeed := 0,
	                                  ix_SafetyOk := #ix_SafetyOk,
	                                  ix_24vOk := #ix_24vOk,
	                                  ix_400vOk := #ix_400vOk,
	                                  ix_HardwareOk := #ix_HardwareOk,
	                                  ix_PECEoS := #iqUDT_WorkstationStatus."630".PEC_Eos.PEC,
	                                  ix_PECBoS := TRUE,
	                                  ix_ExternalRequestHold := FALSE,
	                                  qUDT_HMIStatus => #iqUDT_WorkstationStatus."630".Conveyor,
	                                  qUDT_Status => #iqUDT_WorkstationCommonStatus."630",
	                                  iqUDT_EquipmentControl := #iqUDT_EquipmentControl,
	                                  iqUDT_ConveyorCommand := #iqUDT_WorkstationCommands."630".Conveyor,
	                                  iqUDT_ConveyorInterface := #sUDT_Interface_630,
	                                  iqUDT_HandShakeUp := #sUDT_Handshake_620,
	                                  iqUDT_HandShake := #sUDT_Handshake_630,
	                                  iqUDT_Statistics := #iqUDT_WorkstationStatistics."630".Conveyor);
	            END_REGION

	            REGION MCO
	                #sFB_MCOConveyLinxAixController_630(iUDT_AixConfig := #iUDT_Configuration."630".MCO_M01,
	                                                    iv_AixInputsModule := #iUDT_MotorInput620,
	                                                    ix_24vOk := #ix_24vOk,
	                                                    ix_SimulationModeActive := "DB_Memory".Simulation,
	                                                    ii_MotorPositionId := 2,
	                                                    qUDT_HMIStatus => #iqUDT_WorkstationStatus."630".MCO_M01,
	                                                    iqv_AixOutputsModule := #qUDT_MotorOutput620,
	                                                    iqUDT_ConveyorInterface := #sUDT_Interface_630,
	                                                    iqUDT_MCOStatistics := #iqUDT_WorkstationStatistics."630".MCO_M01);
	            END_REGION
	        END_REGION

	        REGION 640

	            REGION Displacement

	                #sFB_Displacement640(#sUDT_Interface_640);

	            END_REGION

	            REGION MCO
	                #sFB_MCOConveyLinxAixController_640(iUDT_AixConfig := #iUDT_Configuration."640".MCO_M01,
	                                                    iv_AixInputsModule := #iUDT_MotorInput640,
	                                                    ii_PositionSetpoint := #iqUDT_RATPositioning640.Lower.EndPosition,
	                                                    ix_24vOk := #ix_24vOk,
	                                                    ix_SimulationModeActive := "DB_Memory".Simulation,
	                                                    ii_MotorPositionId := 1,
	                                                    ix_StartPositioning := #iqUDT_RATPositioning640.Lower.Start,
	                                                    ix_ResetPosition := #iqUDT_RATPositioning640.Lower.ResetPosition,
	                                                    qUDT_HMIStatus => #iqUDT_WorkstationStatus."640".MCO_M01,
	                                                    qx_Positioned => #iqUDT_RATPositioning640.Lower.Done,
	                                                    iqv_AixOutputsModule := #qUDT_MotorOutput640,
	                                                    iqUDT_ConveyorInterface := #sUDT_Interface_640,
	                                                    iqUDT_MCOStatistics := #iqUDT_WorkstationStatistics."640".MCO_M01);
	            END_REGION


	        END_REGION
	        REGION 641

	            REGION Displacement

	                #sFB_Displacement641(#sUDT_Interface_641);

	            END_REGION

	            REGION RAT


	                #sFB_RightAngledTransfer_641(iUDT_Configuration := #iUDT_Configuration."641".RightAngledTransfer,
	                                             iUDT_LowerConveyorConfiguration := #iUDT_Configuration."640".Conveyor,
	                                             iUDT_UpperConveyorConfiguration := #iUDT_Configuration."641".Conveyor,
	                                             iUDT_PECConfiguration := #iUDT_Configuration."640".PEC_Eos,
	                                             ii_DestinationA := #si_640DestinationA,
	                                             ii_DestinationB := #si_640DestinationB,
	                                             ii_DestinationC := #si_640DestinationC,
	                                             ii_DestinationD := #si_640DestinationD,
	                                             ix_HardwareOk := #ix_HardwareOk,
	                                             ix_400vOk := #ix_400vOk,
	                                             ix_24vOk := #ix_24vOk,
	                                             ix_SafetyOk := #ix_SafetyOk,
	                                             ix_AirPressureOk := #ix_AirPressureOk,
	                                             ix_SectionIsDown := #ix_SectionIsDown641,
	                                             ix_SectionIsUp := #ix_SectionIsUp641,
	                                             ix_ConveyorAAuto := #iqUDT_WorkstationCommonStatus."630".AutoON,
	                                             ix_ConveyorBAuto := #iqUDT_WorkstationCommonStatus."670".AutoON,
	                                             ix_ConveyorCAuto := FALSE,
	                                             ix_ConveyorDAuto := #iqUDT_WorkstationCommonStatus."651".AutoON,
	                                             ix_PEC := #iUDT_MotorInput640.AllSensorPortInputs.LeftSensor,
	                                             ix_ExternalReceiveRequestA := NOT #iqUDT_WorkstationStatus."630".PEC_Eos.PEC,
	                                             ix_ExternalReceiveRequestB := false,
	                                             ix_ExternalReceiveRequestC := false,
	                                             ix_ExternalReceiveRequestD := false,
	                                             ix_PECInfeedA := #iqUDT_WorkstationStatus."630".PEC_Eos.PEC,
	                                             qUDT_HMIRATStatus => #iqUDT_WorkstationStatus."641".RightAngledTransfer,
	                                             qUDT_HMIConveyorStatus => #iqUDT_WorkstationStatus."640".Conveyor,
	                                             qUDT_HMIPECStatus => #iqUDT_WorkstationStatus."640".PEC_Eos,
	                                             qUDT_RATStatus => #iqUDT_WorkstationCommonStatus."641",
	                                             qUDT_ConveyorStatus => #iqUDT_WorkstationCommonStatus."640",
	                                             qx_PopupControl => #qx_PopupControl641,
	                                             iqUDT_EquipmentControl := #iqUDT_EquipmentControl,
	                                             iqUDT_RATCommand := #iqUDT_WorkstationCommands."641".RightAngledTransfer,
	                                             iqUDT_ConveyorCommand := #iqUDT_WorkstationCommands."640".Conveyor,
	                                             iqUDT_RATStatistics := #iqUDT_WorkstationStatistics."641".RightAngledTransfer,
	                                             iqUDT_ConveyorStatistics := #iqUDT_WorkstationStatistics."640".Conveyor,
	                                             iqUDT_PECStatistics := #iqUDT_WorkstationStatistics."640".PEC_Eos,
	                                             iqUDT_HandShakeConveyorA := #sUDT_Handshake_630,
	                                             iqUDT_HandShakeConveyorB := #sUDT_Handshake_640,
	                                             iqUDT_HandShakeConveyorC := #sUDT_HandshakeUp_641,
	                                             iqUDT_HandShakeConveyorD := #sUDT_Handshake_641,
	                                             iqUDT_LowerConveyorInterface := #sUDT_Interface_640,
	                                             iqUDT_UpperConveyorInterface := #sUDT_Interface_641,
	                                             iqUDT_RATPositioning := #iqUDT_RATPositioning640,
	                                             iqUDT_BladeStopEoSInterface := #tUDT_DummyBladeStop,
	                                             iqUDT_BladeStopBoSInterface := #tUDT_DummyBladeStop);

	            END_REGION
	            REGION MCO
	                #sFB_MCOConveyLinxAixController_641(iUDT_AixConfig := #iUDT_Configuration."641".MCO_M01,
	                                                    iv_AixInputsModule := #iUDT_MotorInput640,
	                                                    ix_24vOk := #ix_24vOk,
	                                                    ix_SimulationModeActive := "DB_Memory".Simulation,
	                                                    ii_MotorPositionId := 2,
	                                                    qUDT_HMIStatus => #iqUDT_WorkstationStatus."641".MCO_M01,
	                                                    iqv_AixOutputsModule := #qUDT_MotorOutput640,
	                                                    iqUDT_ConveyorInterface := #sUDT_Interface_641,
	                                                    iqUDT_MCOStatistics := #iqUDT_WorkstationStatistics."641".MCO_M01);
	            END_REGION
	        END_REGION

	        REGION 650

	            REGION Displacement

	                #sFB_Displacement650(#sUDT_Interface_650);

	            END_REGION

	            REGION MCO
	                #sFB_MCOConveyLinxAixController_650(iUDT_AixConfig := #iUDT_Configuration."650".MCO_M01,
	                                                    iv_AixInputsModule := #iUDT_MotorInput650,
	                                                    ix_24vOk := #ix_24vOk,
	                                                    ix_SimulationModeActive := "DB_Memory".Simulation,
	                                                    ii_MotorPositionId := 1,
	                                                    qUDT_HMIStatus => #iqUDT_WorkstationStatus."650".MCO_M01,
	                                                    iqv_AixOutputsModule := #qUDT_MotorOutput650,
	                                                    iqUDT_ConveyorInterface := #sUDT_Interface_650,
	                                                    iqUDT_MCOStatistics := #iqUDT_WorkstationStatistics."650".MCO_M01);
	            END_REGION

	        END_REGION
	        REGION 651

	            REGION Displacement

	                #sFB_Displacement651(#sUDT_Interface_651);

	            END_REGION

	            REGION RAT

	                #sFB_RightAngledTransfer_651(iUDT_Configuration := #iUDT_Configuration."651".RightAngledTransfer,
	                                             iUDT_LowerConveyorConfiguration := #iUDT_Configuration."650".Conveyor,
	                                             iUDT_UpperConveyorConfiguration := #iUDT_Configuration."651".Conveyor,
	                                             iUDT_PECConfiguration := #iUDT_Configuration."650".PEC_Eos,
	                                             ii_DestinationA := #si_650DestinationA,
	                                             ii_DestinationB := #si_650DestinationB,
	                                             ii_DestinationC := #si_650DestinationC,
	                                             ii_DestinationD := #si_650DestinationD,
	                                             ix_HardwareOk := #ix_HardwareOk,
	                                             ix_400vOk := #ix_400vOk,
	                                             ix_24vOk := #ix_24vOk,
	                                             ix_SafetyOk := #ix_SafetyOk,
	                                             ix_AirPressureOk := #ix_AirPressureOk,
	                                             ix_SectionIsDown := #ix_SectionIsDown651,
	                                             ix_SectionIsUp := #ix_SectionIsUp651,
	                                             ix_ConveyorAAuto := false,
	                                             ix_ConveyorBAuto := #iqUDT_WorkstationCommonStatus."660".AutoON,
	                                             ix_ConveyorCAuto := #iqUDT_WorkstationCommonStatus."641".AutoON,
	                                             ix_ConveyorDAuto := false,
	                                             ix_PEC := #iUDT_MotorInput650.AllSensorPortInputs.LeftSensor,
	                                             ix_ExternalReceiveRequestA := false,
	                                             ix_ExternalReceiveRequestB := false,
	                                             ix_ExternalReceiveRequestC := #sFB_RightAngledTransfer_641.qx_ExternalSendRequestD,
	                                             ix_ExternalReceiveRequestD := false,
	                                             ix_PECInfeedC := #iqUDT_WorkstationStatus."640".PEC_Eos.PEC,
	                                             qUDT_HMIRATStatus => #iqUDT_WorkstationStatus."651".RightAngledTransfer,
	                                             qUDT_HMIConveyorStatus => #iqUDT_WorkstationStatus."650".Conveyor,
	                                             qUDT_HMIPECStatus => #iqUDT_WorkstationStatus."650".PEC_Eos,
	                                             qUDT_RATStatus => #iqUDT_WorkstationCommonStatus."651",
	                                             qUDT_ConveyorStatus => #iqUDT_WorkstationCommonStatus."650",
	                                             qx_PopupControl => #qx_PopupControl651,
	                                             iqUDT_EquipmentControl := #iqUDT_EquipmentControl,
	                                             iqUDT_RATCommand := #iqUDT_WorkstationCommands."651".RightAngledTransfer,
	                                             iqUDT_ConveyorCommand := #iqUDT_WorkstationCommands."650".Conveyor,
	                                             iqUDT_RATStatistics := #iqUDT_WorkstationStatistics."651".RightAngledTransfer,
	                                             iqUDT_ConveyorStatistics := #iqUDT_WorkstationStatistics."650".Conveyor,
	                                             iqUDT_PECStatistics := #iqUDT_WorkstationStatistics."650".PEC_Eos,
	                                             iqUDT_HandShakeConveyorA := #tUDT_dummyHandshake,
	                                             iqUDT_HandShakeConveyorB := #sUDT_Handshake_650,
	                                             iqUDT_HandShakeConveyorC := #sUDT_Handshake_641,
	                                             iqUDT_HandShakeConveyorD := #tUDT_dummyHandshake,
	                                             iqUDT_LowerConveyorInterface := #sUDT_Interface_650,
	                                             iqUDT_UpperConveyorInterface := #sUDT_Interface_651,
	                                             iqUDT_RATPositioning := #iqUDT_RATPositioning650,
	                                             iqUDT_BladeStopEoSInterface := #tUDT_DummyBladeStop,
	                                             iqUDT_BladeStopBoSInterface := #tUDT_DummyBladeStop);

	            END_REGION

	            REGION MCO
	                #sFB_MCOConveyLinxAixController_651(iUDT_AixConfig := #iUDT_Configuration."651".MCO_M01,
	                                                    iv_AixInputsModule := #iUDT_MotorInput650,
	                                                    ii_PositionSetpoint := #iqUDT_RATPositioning650.Upper.EndPosition,
	                                                    ix_24vOk := #ix_24vOk,
	                                                    ix_SimulationModeActive := "DB_Memory".Simulation,
	                                                    ii_MotorPositionId := 2,
	                                                    ix_StartPositioning := #iqUDT_RATPositioning650.Upper.Start,
	                                                    ix_ResetPosition := #iqUDT_RATPositioning650.Upper.ResetPosition,
	                                                    qUDT_HMIStatus => #iqUDT_WorkstationStatus."651".MCO_M01,
	                                                    qx_Positioned => #iqUDT_RATPositioning650.Upper.Done,
	                                                    iqv_AixOutputsModule := #qUDT_MotorOutput650,
	                                                    iqUDT_ConveyorInterface := #sUDT_Interface_651,
	                                                    iqUDT_MCOStatistics := #iqUDT_WorkstationStatistics."651".MCO_M01);
	            END_REGION
	        END_REGION

	        REGION 660

	            REGION Displacement

	                #sFB_Displacement660(#sUDT_Interface_660);

	            END_REGION

	            REGION MCO
	                #sFB_MCOConveyLinxAixController_660(iUDT_AixConfig := #iUDT_Configuration."660".MCO_M01,
	                                                    iv_AixInputsModule := #iUDT_MotorInput660,
	                                                    ii_PositionSetpoint := #iqUDT_RATPositioning660.Lower.EndPosition,
	                                                    ix_24vOk := #ix_24vOk,
	                                                    ix_SimulationModeActive := "DB_Memory".Simulation,
	                                                    ii_MotorPositionId := 1,
	                                                    ix_StartPositioning := #iqUDT_RATPositioning660.Lower.Start,
	                                                    ix_ResetPosition := #iqUDT_RATPositioning660.Lower.ResetPosition,
	                                                    qUDT_HMIStatus => #iqUDT_WorkstationStatus."660".MCO_M01,
	                                                    qx_Positioned => #iqUDT_RATPositioning660.Lower.Done,
	                                                    iqv_AixOutputsModule := #qUDT_MotorOutput660,
	                                                    iqUDT_ConveyorInterface := #sUDT_Interface_660,
	                                                    iqUDT_MCOStatistics := #iqUDT_WorkstationStatistics."660".MCO_M01);
	            END_REGION

	        END_REGION
	        REGION 661

	            REGION Displacement

	                #sFB_Displacement661(#sUDT_Interface_661);

	            END_REGION

	            REGION RAT

	                #sFB_RightAngledTransfer_661(iUDT_Configuration := #iUDT_Configuration."661".RightAngledTransfer,
	                                             iUDT_LowerConveyorConfiguration := #iUDT_Configuration."660".Conveyor,
	                                             iUDT_UpperConveyorConfiguration := #iUDT_Configuration."661".Conveyor,
	                                             iUDT_PECConfiguration := #iUDT_Configuration."660".PEC_Eos,
	                                             ii_DestinationA := #si_660DestinationA,
	                                             ii_DestinationB := #si_660DestinationB,
	                                             ii_DestinationC := #si_660DestinationC,
	                                             ii_DestinationD := #si_660DestinationD,
	                                             ix_HardwareOk := #ix_HardwareOk,
	                                             ix_400vOk := #ix_400vOk,
	                                             ix_24vOk := #ix_24vOk,
	                                             ix_SafetyOk := #ix_SafetyOk,
	                                             ix_AirPressureOk := #ix_AirPressureOk,
	                                             ix_SectionIsDown := #ix_SectionIsDown661,
	                                             ix_SectionIsUp := #ix_SectionIsUp661,
	                                             ix_ConveyorAAuto := #iqUDT_WorkstationCommonStatus."650".AutoON,
	                                             ix_ConveyorBAuto := #iqUDT_WorkstationCommonStatus."680".AutoON,
	                                             ix_ConveyorCAuto := #iqUDT_WorkstationCommonStatus."671".AutoON,
	                                             ix_ConveyorDAuto := false,
	                                             ix_PEC := #iUDT_MotorInput660.AllSensorPortInputs.LeftSensor,
	                                             ix_ExternalReceiveRequestA := #sFB_RightAngledTransfer_651.qx_ExternalSendRequestB AND (#sx_ActiveRequest680 OR #sx_ClearLeftStation),
	                                             ix_ExternalReceiveRequestB := (#sx_TransferOut680 OR #sx_ClearLeftStation) AND NOT #iqUDT_WorkstationStatus."680".PEC_Eos.PEC,
	                                             ix_ExternalReceiveRequestC := false,
	                                             ix_ExternalReceiveRequestD := false,
	                                             ix_PECInfeedA := #iqUDT_WorkstationStatus."650".PEC_Eos.PEC,
	                                             ix_PECInfeedB := #iqUDT_WorkstationStatus."680".PEC_Eos.PEC,
	                                             qUDT_HMIRATStatus => #iqUDT_WorkstationStatus."661".RightAngledTransfer,
	                                             qUDT_HMIConveyorStatus => #iqUDT_WorkstationStatus."660".Conveyor,
	                                             qUDT_HMIPECStatus => #iqUDT_WorkstationStatus."660".PEC_Eos,
	                                             qUDT_RATStatus => #iqUDT_WorkstationCommonStatus."661",
	                                             qUDT_ConveyorStatus => #iqUDT_WorkstationCommonStatus."660",
	                                             qx_PopupControl => #qx_PopupControl661,
	                                             iqUDT_EquipmentControl := #iqUDT_EquipmentControl,
	                                             iqUDT_RATCommand := #iqUDT_WorkstationCommands."661".RightAngledTransfer,
	                                             iqUDT_ConveyorCommand := #iqUDT_WorkstationCommands."660".Conveyor,
	                                             iqUDT_RATStatistics := #iqUDT_WorkstationStatistics."661".RightAngledTransfer,
	                                             iqUDT_ConveyorStatistics := #iqUDT_WorkstationStatistics."660".Conveyor,
	                                             iqUDT_PECStatistics := #iqUDT_WorkstationStatistics."660".PEC_Eos,
	                                             iqUDT_HandShakeConveyorA := #sUDT_Handshake_650,
	                                             iqUDT_HandShakeConveyorB := #sUDT_Handshake_660,
	                                             iqUDT_HandShakeConveyorC := #sUDT_HandshakeUp_661,
	                                             iqUDT_HandShakeConveyorD := #tUDT_dummyHandshake,
	                                             iqUDT_LowerConveyorInterface := #sUDT_Interface_660,
	                                             iqUDT_UpperConveyorInterface := #sUDT_Interface_661,
	                                             iqUDT_RATPositioning := #iqUDT_RATPositioning660,
	                                             iqUDT_BladeStopEoSInterface := #tUDT_DummyBladeStop,
	                                             iqUDT_BladeStopBoSInterface := #tUDT_DummyBladeStop);

	            END_REGION

	            REGION MCO
	                #sFB_MCOConveyLinxAixController_661(iUDT_AixConfig := #iUDT_Configuration."661".MCO_M01,
	                                                    iv_AixInputsModule := #iUDT_MotorInput660,
	                                                    ix_24vOk := #ix_24vOk,
	                                                    ix_SimulationModeActive := "DB_Memory".Simulation,
	                                                    ii_MotorPositionId := 2,
	                                                    qUDT_HMIStatus => #iqUDT_WorkstationStatus."661".MCO_M01,
	                                                    iqv_AixOutputsModule := #qUDT_MotorOutput660,
	                                                    iqUDT_ConveyorInterface := #sUDT_Interface_661,
	                                                    iqUDT_MCOStatistics := #iqUDT_WorkstationStatistics."661".MCO_M01);
	            END_REGION
	        END_REGION

	        REGION 670

	            REGION Displacement

	                #sFB_Displacement670(#sUDT_Interface_670);

	            END_REGION

	            REGION MCO
	                #sFB_MCOConveyLinxAixController_670(iUDT_AixConfig := #iUDT_Configuration."670".MCO_M01,
	                                                    iv_AixInputsModule := #iUDT_MotorInput670,
	                                                    ii_PositionSetpoint := #iqUDT_RATPositioning670.Lower.EndPosition,
	                                                    ix_24vOk := #ix_24vOk,
	                                                    ix_SimulationModeActive := "DB_Memory".Simulation,
	                                                    ii_MotorPositionId := 1,
	                                                    ix_StartPositioning := #iqUDT_RATPositioning670.Lower.Start,
	                                                    ix_ResetPosition := #iqUDT_RATPositioning670.Lower.ResetPosition,
	                                                    qUDT_HMIStatus => #iqUDT_WorkstationStatus."670".MCO_M01,
	                                                    qx_Positioned => #iqUDT_RATPositioning670.Lower.Done,
	                                                    iqv_AixOutputsModule := #qUDT_MotorOutput670,
	                                                    iqUDT_ConveyorInterface := #sUDT_Interface_670,
	                                                    iqUDT_MCOStatistics := #iqUDT_WorkstationStatistics."670".MCO_M01);
	            END_REGION

	        END_REGION

	        REGION 671

	            REGION Displacement

	                #sFB_Displacement671(#sUDT_Interface_671);

	            END_REGION

	            REGION RAT

	                #sFB_RightAngledTransfer_671(iUDT_Configuration := #iUDT_Configuration."671".RightAngledTransfer,
	                                             iUDT_LowerConveyorConfiguration := #iUDT_Configuration."670".Conveyor,
	                                             iUDT_UpperConveyorConfiguration := #iUDT_Configuration."671".Conveyor,
	                                             iUDT_PECConfiguration := #iUDT_Configuration."670".PEC_Eos,
	                                             ii_DestinationA := #si_670DestinationA,
	                                             ii_DestinationB := #si_670DestinationB,
	                                             ii_DestinationC := #si_670DestinationC,
	                                             ii_DestinationD := #si_670DestinationD,
	                                             ix_HardwareOk := #ix_HardwareOk,
	                                             ix_400vOk := #ix_400vOk,
	                                             ix_24vOk := #ix_24vOk,
	                                             ix_SafetyOk := #ix_SafetyOk,
	                                             ix_AirPressureOk := #ix_AirPressureOk,
	                                             ix_SectionIsDown := #ix_SectionIsDown671,
	                                             ix_SectionIsUp := #ix_SectionIsUp671,
	                                             ix_ConveyorAAuto := #iqUDT_WorkstationCommonStatus."630".AutoON,
	                                             ix_ConveyorBAuto := #iqUDT_WorkstationCommonStatus."670".AutoON,
	                                             ix_ConveyorCAuto := FALSE,
	                                             ix_ConveyorDAuto := #iqUDT_WorkstationCommonStatus."650".AutoON,
	                                             ix_PEC := #iUDT_MotorInput670.AllSensorPortInputs.LeftSensor,
	                                             ix_ExternalReceiveRequestA := #sFB_RightAngledTransfer_641.qx_ExternalSendRequestB,
	                                             ix_ExternalReceiveRequestB := (#sx_TransferOut690 OR #sx_ClearLeftStation) AND NOT #iqUDT_WorkstationStatus."690".PEC_Eos.PEC,
	                                             ix_ExternalReceiveRequestC := false,
	                                             ix_ExternalReceiveRequestD := #sFB_RightAngledTransfer_661.qx_ExternalSendRequestC,
	                                             ix_PECInfeedA := #iqUDT_WorkstationStatus."640".PEC_Eos.PEC,
	                                             ix_PECInfeedB := #iqUDT_WorkstationStatus."690".PEC_Eos.PEC,
	                                             ix_PECInfeedD := #iqUDT_WorkstationStatus."660".PEC_Eos.PEC,
	                                             qUDT_HMIRATStatus => #iqUDT_WorkstationStatus."671".RightAngledTransfer,
	                                             qUDT_HMIConveyorStatus => #iqUDT_WorkstationStatus."670".Conveyor,
	                                             qUDT_HMIPECStatus => #iqUDT_WorkstationStatus."670".PEC_Eos,
	                                             qUDT_RATStatus => #iqUDT_WorkstationCommonStatus."671",
	                                             qUDT_ConveyorStatus => #iqUDT_WorkstationCommonStatus."670",
	                                             qx_PopupControl => #qx_PopupControl671,
	                                             iqUDT_EquipmentControl := #iqUDT_EquipmentControl,
	                                             iqUDT_RATCommand := #iqUDT_WorkstationCommands."671".RightAngledTransfer,
	                                             iqUDT_ConveyorCommand := #iqUDT_WorkstationCommands."670".Conveyor,
	                                             iqUDT_RATStatistics := #iqUDT_WorkstationStatistics."671".RightAngledTransfer,
	                                             iqUDT_ConveyorStatistics := #iqUDT_WorkstationStatistics."670".Conveyor,
	                                             iqUDT_PECStatistics := #iqUDT_WorkstationStatistics."670".PEC_Eos,
	                                             iqUDT_HandShakeConveyorA := #sUDT_Handshake_640,
	                                             iqUDT_HandShakeConveyorB := #sUDT_Handshake_670,
	                                             iqUDT_HandShakeConveyorC := #sUDT_HandshakeUp_671,
	                                             iqUDT_HandShakeConveyorD := #sUDT_HandshakeUp_661,
	                                             iqUDT_LowerConveyorInterface := #sUDT_Interface_670,
	                                             iqUDT_UpperConveyorInterface := #sUDT_Interface_671,
	                                             iqUDT_RATPositioning := #iqUDT_RATPositioning670,
	                                             iqUDT_BladeStopEoSInterface := #tUDT_DummyBladeStop,
	                                             iqUDT_BladeStopBoSInterface := #tUDT_DummyBladeStop);

	            END_REGION

	            REGION MCO
	                #sFB_MCOConveyLinxAixController_671(iUDT_AixConfig := #iUDT_Configuration."671".MCO_M01,
	                                                    iv_AixInputsModule := #iUDT_MotorInput670,
	                                                    ii_PositionSetpoint := #iqUDT_RATPositioning670.Upper.EndPosition,
	                                                    ix_24vOk := #ix_24vOk,
	                                                    ix_SimulationModeActive := "DB_Memory".Simulation,
	                                                    ii_MotorPositionId := 2,
	                                                    ix_StartPositioning := #iqUDT_RATPositioning670.Upper.Start,
	                                                    ix_ResetPosition := #iqUDT_RATPositioning670.Upper.ResetPosition,
	                                                    qUDT_HMIStatus => #iqUDT_WorkstationStatus."671".MCO_M01,
	                                                    qx_Positioned => #iqUDT_RATPositioning670.Upper.Done,
	                                                    iqv_AixOutputsModule := #qUDT_MotorOutput670,
	                                                    iqUDT_ConveyorInterface := #sUDT_Interface_671,
	                                                    iqUDT_MCOStatistics := #iqUDT_WorkstationStatistics."671".MCO_M01);
	            END_REGION
	        END_REGION

	        REGION 680

	            REGION Displacement

	                #sFB_Displacement680(#sUDT_Interface_680);

	            END_REGION

	            REGION Tracking

	                #sFB_Tracking_680(iUDT_ConveyorCommonConfiguration := #iUDT_Configuration."680".Conveyor.Common,
	                                  iqa_TrackingData := #sa_TrackingArray_680,
	                                  iqUDT_ConveyorInterface := #sUDT_Interface_680,
	                                  iqUDT_HandshakeUp := #sUDT_Handshake_660,
	                                  iqUDT_Handshake := #sUDT_Handshake_680);
	            END_REGION

	            REGION EOS

	                #sFB_PECUpdate_680(iUDT_PECUpdateConfiguration := #iUDT_Configuration."680".PEC_Eos,
	                                   iUDT_ConveyorCommonConfiguration := #iUDT_Configuration."680".Conveyor.Common,
	                                   ix_PEC := #iUDT_MotorInput680.AllSensorPortInputs.LeftSensor,
	                                   ix_TeachingMode := FALSE,
	                                   qUDT_Status => #iqUDT_WorkstationStatus."680".PEC_Eos,
	                                   qi_GINwrite => #ti_dummy,
	                                   qx_PECFiltered => #tx_dummy,
	                                   iqa_TrackingData := #sa_TrackingArray_680,
	                                   iqUDT_ConveyorInterface := #sUDT_Interface_680,
	                                   iqUDT_UnknownGINRange := #iqUDT_UnknownGINRange,
	                                   iqUDT_FifoHeader := "DB_FIFOLostGIN".Header,
	                                   iqa_FifoData := "DB_FIFOLostGIN".Data,
	                                   iqUDT_Statistics := #iqUDT_WorkstationStatistics."680".PEC_Eos);

	            END_REGION

	            REGION Conveyor

	                #sUDT_Handshake_680.RTR := #iqUDT_WorkstationStatus."680".PEC_Eos.PEC;

	                #sFB_Conveyor_680(iUDT_ConveyorConfiguration := #iUDT_Configuration."680".Conveyor,
	                                  idi_PECEoSDistance := #iUDT_Configuration."680".PEC_Eos.Distance,
	                                  idi_PECBoSDistance := 0,
	                                  ii_ExternalSpeed := 0,
	                                  ix_SafetyOk := #ix_SafetyOk,
	                                  ix_24vOk := #ix_24vOk,
	                                  ix_400vOk := #ix_400vOk,
	                                  ix_HardwareOk := #ix_HardwareOk,
	                                  ix_ReverseDirection := #sx_DirectionChange680,
	                                  ix_PECEoS := #iqUDT_WorkstationStatus."680".PEC_Eos.PEC,
	                                  ix_PECBoS := TRUE,
	                                  ix_ExternalRequestHold := false,
	                                  qUDT_HMIStatus => #iqUDT_WorkstationStatus."680".Conveyor,
	                                  qUDT_Status => #iqUDT_WorkstationCommonStatus."680",
	                                  iqUDT_EquipmentControl := #iqUDT_EquipmentControl,
	                                  iqUDT_ConveyorCommand := #iqUDT_WorkstationCommands."680".Conveyor,
	                                  iqUDT_ConveyorInterface := #sUDT_Interface_680,
	                                  iqUDT_HandShakeUp := #sUDT_Handshake_660,
	                                  iqUDT_HandShake := #sUDT_Handshake_680,
	                                  iqUDT_Statistics := #iqUDT_WorkstationStatistics."680".Conveyor);
	            END_REGION

	            REGION MCO
	                #sFB_MCOConveyLinxAixController_680(iUDT_AixConfig := #iUDT_Configuration."680".MCO_M01,
	                                                    iv_AixInputsModule := #iUDT_MotorInput680,
	                                                    ix_24vOk := #ix_24vOk,
	                                                    ix_SimulationModeActive := "DB_Memory".Simulation,
	                                                    ii_MotorPositionId := 1,
	                                                    qUDT_HMIStatus => #iqUDT_WorkstationStatus."680".MCO_M01,
	                                                    iqv_AixOutputsModule := #qUDT_MotorOutput680,
	                                                    iqUDT_ConveyorInterface := #sUDT_Interface_680,
	                                                    iqUDT_MCOStatistics := #iqUDT_WorkstationStatistics."680".MCO_M01);
	            END_REGION

	        END_REGION

	        REGION 690

	            REGION Displacement

	                #sFB_Displacement690(#sUDT_Interface_690);

	            END_REGION

	            REGION Tracking

	                #sFB_Tracking_690(iUDT_ConveyorCommonConfiguration := #iUDT_Configuration."690".Conveyor.Common,
	                                  iqa_TrackingData := #sa_TrackingArray_690,
	                                  iqUDT_ConveyorInterface := #sUDT_Interface_690,
	                                  iqUDT_HandshakeUp := #sUDT_Handshake_670,
	                                  iqUDT_Handshake := #sUDT_Handshake_690);
	            END_REGION

	            REGION EOS

	                #sFB_PECUpdate_690(iUDT_PECUpdateConfiguration := #iUDT_Configuration."690".PEC_Eos,
	                                   iUDT_ConveyorCommonConfiguration := #iUDT_Configuration."690".Conveyor.Common,
	                                   ix_PEC := #iUDT_MotorInput690.AllSensorPortInputs.LeftSensor,
	                                   ix_TeachingMode := FALSE,
	                                   qUDT_Status => #iqUDT_WorkstationStatus."690".PEC_Eos,
	                                   qi_GINwrite => #ti_dummy,
	                                   qx_PECFiltered => #tx_dummy,
	                                   iqa_TrackingData := #sa_TrackingArray_690,
	                                   iqUDT_ConveyorInterface := #sUDT_Interface_690,
	                                   iqUDT_UnknownGINRange := #iqUDT_UnknownGINRange,
	                                   iqUDT_FifoHeader := "DB_FIFOLostGIN".Header,
	                                   iqa_FifoData := "DB_FIFOLostGIN".Data,
	                                   iqUDT_Statistics := #iqUDT_WorkstationStatistics."690".PEC_Eos);

	            END_REGION

	            REGION Conveyor

	                #sUDT_Handshake_690.RTR := #iqUDT_WorkstationStatus."690".PEC_Eos.PEC;


	                #sFB_Conveyor_690(iUDT_ConveyorConfiguration := #iUDT_Configuration."690".Conveyor,
	                                  idi_PECEoSDistance := #iUDT_Configuration."690".PEC_Eos.Distance,
	                                  idi_PECBoSDistance := 0,
	                                  ii_ExternalSpeed := 0,
	                                  ix_SafetyOk := #ix_SafetyOk,
	                                  ix_24vOk := #ix_24vOk,
	                                  ix_400vOk := #ix_400vOk,
	                                  ix_HardwareOk := #ix_HardwareOk,
	                                  ix_ReverseDirection := #sx_DirectionChange690,
	                                  ix_PECEoS := #iqUDT_WorkstationStatus."690".PEC_Eos.PEC,
	                                  ix_PECBoS := TRUE,
	                                  ix_ExternalRequestHold := FALSE,
	                                  qUDT_HMIStatus => #iqUDT_WorkstationStatus."690".Conveyor,
	                                  qUDT_Status => #iqUDT_WorkstationCommonStatus."690",
	                                  iqUDT_EquipmentControl := #iqUDT_EquipmentControl,
	                                  iqUDT_ConveyorCommand := #iqUDT_WorkstationCommands."690".Conveyor,
	                                  iqUDT_ConveyorInterface := #sUDT_Interface_690,
	                                  iqUDT_HandShakeUp := #sUDT_Handshake_670,
	                                  iqUDT_HandShake := #sUDT_Handshake_690,
	                                  iqUDT_Statistics := #iqUDT_WorkstationStatistics."690".Conveyor);
	            END_REGION

	            REGION MCO
	                #sFB_MCOConveyLinxAixController_690(iUDT_AixConfig := #iUDT_Configuration."690".MCO_M01,
	                                                    iv_AixInputsModule := #iUDT_MotorInput690,
	                                                    ix_24vOk := #ix_24vOk,
	                                                    ix_SimulationModeActive := "DB_Memory".Simulation,
	                                                    ii_MotorPositionId := 1,
	                                                    qUDT_HMIStatus => #iqUDT_WorkstationStatus."690".MCO_M01,
	                                                    iqv_AixOutputsModule := #qUDT_MotorOutput690,
	                                                    iqUDT_ConveyorInterface := #sUDT_Interface_690,
	                                                    iqUDT_MCOStatistics := #iqUDT_WorkstationStatistics."690".MCO_M01);
	            END_REGION
	        END_REGION

	        REGION 530

	            REGION Displacement

	                #sFB_Displacement530(#sUDT_Interface_530);

	            END_REGION

	            REGION Tracking

	                #sFB_Tracking_530(iUDT_ConveyorCommonConfiguration := #iUDT_Configuration."530".Conveyor.Common,
	                                  iqa_TrackingData := #sa_TrackingArray_530,
	                                  iqUDT_ConveyorInterface := #sUDT_Interface_530,
	                                  iqUDT_HandshakeUp := #sUDT_Handshake_530,
	                                  iqUDT_Handshake := #sUDT_Handshake_530);
	            END_REGION

	            REGION EOS

	                #sFB_PECUpdate_530(iUDT_PECUpdateConfiguration := #iUDT_Configuration."530".PEC_Eos,
	                                   iUDT_ConveyorCommonConfiguration := #iUDT_Configuration."530".Conveyor.Common,
	                                   ix_PEC := #iUDT_MotorInput530.AllSensorPortInputs.LeftSensor,
	                                   ix_TeachingMode := FALSE,
	                                   qUDT_Status => #iqUDT_WorkstationStatus."530".PEC_Eos,
	                                   qi_GINwrite => #ti_dummy,
	                                   qx_PECFiltered => #tx_dummy,
	                                   iqa_TrackingData := #sa_TrackingArray_530,
	                                   iqUDT_ConveyorInterface := #sUDT_Interface_530,
	                                   iqUDT_UnknownGINRange := #iqUDT_UnknownGINRange,
	                                   iqUDT_FifoHeader := "DB_FIFOLostGIN".Header,
	                                   iqa_FifoData := "DB_FIFOLostGIN".Data,
	                                   iqUDT_Statistics := #iqUDT_WorkstationStatistics."530".PEC_Eos);

	            END_REGION

	            REGION Conveyor
	                #sUDT_Handshake_530.RTR := #sUDT_Handshake_530.RTR OR #iqUDT_WorkstationStatus."530".PEC_Eos.PEC;

	                #sFB_Conveyor_530(iUDT_ConveyorConfiguration := #iUDT_Configuration."530".Conveyor,
	                                  idi_PECEoSDistance := #iUDT_Configuration."530".PEC_Eos.Distance,
	                                  idi_PECBoSDistance := 0,
	                                  ii_ExternalSpeed := 0,
	                                  ix_SafetyOk := #ix_SafetyOk,
	                                  ix_24vOk := #ix_24vOk,
	                                  ix_400vOk := #ix_400vOk,
	                                  ix_HardwareOk := #ix_HardwareOk,
	                                  ix_PECEoS := #iqUDT_WorkstationStatus."530".PEC_Eos.PEC,
	                                  ix_PECBoS := TRUE,
	                                  ix_ExternalRequestHold := #sx_Hold530,
	                                  qUDT_HMIStatus => #iqUDT_WorkstationStatus."530".Conveyor,
	                                  qUDT_Status => #iqUDT_WorkstationCommonStatus."530",
	                                  iqUDT_EquipmentControl := #iqUDT_EquipmentControl,
	                                  iqUDT_ConveyorCommand := #iqUDT_WorkstationCommands."530".Conveyor,
	                                  iqUDT_ConveyorInterface := #sUDT_Interface_530,
	                                  iqUDT_HandShakeUp := #sUDT_Handshake_530,
	                                  iqUDT_HandShake := #sUDT_Handshake_530,
	                                  iqUDT_Statistics := #iqUDT_WorkstationStatistics."530".Conveyor);
	            END_REGION

	            REGION MCO
	                #sFB_MCOConveyLinxAixController_530(iUDT_AixConfig := #iUDT_Configuration."530".MCO_M01,
	                                                    iv_AixInputsModule := #iUDT_MotorInput530,
	                                                    ix_24vOk := #ix_24vOk,
	                                                    ix_SimulationModeActive := "DB_Memory".Simulation,
	                                                    ii_MotorPositionId := 1,
	                                                    qUDT_HMIStatus => #iqUDT_WorkstationStatus."530".MCO_M01,
	                                                    iqv_AixOutputsModule := #qUDT_MotorOutput530,
	                                                    iqUDT_ConveyorInterface := #sUDT_Interface_530,
	                                                    iqUDT_MCOStatistics := #iqUDT_WorkstationStatistics."530".MCO_M01);
	            END_REGION
	        END_REGION

	        REGION 540

	            REGION Displacement

	                #sFB_Displacement540(#sUDT_Interface_540);

	            END_REGION

	            REGION MCO
	                #sFB_MCOConveyLinxAixController_540(iUDT_AixConfig := #iUDT_Configuration."540".MCO_M01,
	                                                    iv_AixInputsModule := #iUDT_MotorInput540,
	                                                    ii_PositionSetpoint := #iqUDT_RATPositioning540.Lower.EndPosition,
	                                                    ix_24vOk := #ix_24vOk,
	                                                    ix_SimulationModeActive := "DB_Memory".Simulation,
	                                                    ii_MotorPositionId := 1,
	                                                    ix_StartPositioning := #iqUDT_RATPositioning540.Lower.Start,
	                                                    ix_ResetPosition := #iqUDT_RATPositioning540.Lower.ResetPosition,
	                                                    qUDT_HMIStatus => #iqUDT_WorkstationStatus."540".MCO_M01,
	                                                    qx_Positioned => #iqUDT_RATPositioning540.Lower.Done,
	                                                    iqv_AixOutputsModule := #qUDT_MotorOutput540,
	                                                    iqUDT_ConveyorInterface := #sUDT_Interface_540,
	                                                    iqUDT_MCOStatistics := #iqUDT_WorkstationStatistics."540".MCO_M01);
	            END_REGION

	        END_REGION
	        REGION 541

	            REGION Displacement

	                #sFB_Displacement541(#sUDT_Interface_541);

	            END_REGION

	            REGION RAT

